// TIA Portal V17 export
// export: Created 2022-07-20T07:02:31.7533265Z, ExportSetting WithDefaults, DisplayName Totally Integrated Automation Portal, DisplayVersion V17, DisplayName TIA Portal Openness, DisplayVersion V17, DisplayName TIA Portal Version Control Interface, DisplayVersion V17, DisplayName SINAMICS Startdrive Advanced, DisplayVersion V17, DisplayName SINAMICS Startdrive G130, G150, S120, S150, SINAMICS MV, S210, DisplayVersion V17, DisplayName SINAMICS Startdrive G110M, G120, G120C, G120D, G120P, G115D, DisplayVersion V17, DisplayName STEP 7 Professional, DisplayVersion V17, DisplayName STEP 7 Safety, DisplayVersion V17, DisplayName WinCC Advanced, DisplayVersion V17
FUNCTION_BLOCK "FB11005_SheetEdgeDetection"   // FB11005, LAD
TITLE = Manage sheet edge detection
{ S7_Optimized_Access := 'TRUE' }
VERSION : 0.1
// stored: AutoNumber false, IsIECCheckEnabled false, IsRetainMemResEnabled false, MemoryReserve 100, SetENOAutomatically false, UDAEnableTagReadback false
   VAR_INPUT
      Enable { ExternalAccessible := 'False'; ExternalVisible := 'False'; ExternalWritable := 'False'} : Bool;
      Reset { ExternalAccessible := 'False'; ExternalVisible := 'False'; ExternalWritable := 'False'} : Bool;
      GapDrumSensor { ExternalAccessible := 'False'; ExternalVisible := 'False'; ExternalWritable := 'False'} : Real;
      GapBetweenSheet : Real;
   END_VAR
   VAR_OUTPUT
      Error { ExternalAccessible := 'False'; ExternalVisible := 'False'; ExternalWritable := 'False'} : Bool;
      ErrorSheetTooClose : Bool;
      WarningSheetTooClose : Bool;
      StartSheetPosition { ExternalAccessible := 'False'; ExternalVisible := 'False'; ExternalWritable := 'False'} : LReal;
      SheetDetected { ExternalAccessible := 'False'; ExternalVisible := 'False'; ExternalWritable := 'False'} : Bool;
      SheetGap : LReal;
      SensorActivated : Bool;
   END_VAR
   VAR_IN_OUT
      FilmDrumSensor : TO_MeasuringInput;
   END_VAR
   VAR
      R_TRIG_FilmDrumSensor { S7_SetPoint := 'True'} : R_TRIG;
      statFilmDrumPosition { S7_SetPoint := 'True'} : LReal;
      statFilmDrumPositionOld : LReal;
      statErrorMC : Bool;
      statJam : Bool;
      statOutfeedPosition : LReal;
      statStackerPosition : LReal;
      instMC_MEASURINGINPUT { S7_SetPoint := 'True'} : MC_MEASURINGINPUT;
   END_VAR
BEGIN

REGION Network 1 (SCL): Comments
   //==========================================================================================
   // SIEMENS SAS      RC-FR DI FA APC
   //------------------------------------------------------------------------------------------
   // Restrictions:    TIA V16 and more
   // Requirements:    S7-1500 + MGI library
   // Functionality:   This function block get position value of sheet edge 
   //------------------------------------------------------------------------------------------
   // Change log table:
   // Version      Date        Expert in charge    Changes applied
   // 01.00.01     09.06.2020  RTO                 First released version
   //==========================================================================================
END_REGION

REGION Network 2 (SCL): First Scan
   IF "FirstScan" THEN

       // Output
       #Error := FALSE;
       #SheetDetected := FALSE;
       #StartSheetPosition := 0.0;

       // Static
       #statFilmDrumPosition := 0.0;
       #statFilmDrumPositionOld := 0.0;
       #statErrorMC := FALSE;
       #statJam := FALSE;
       #statOutfeedPosition := 0.0;
       #statStackerPosition := 0.0;

   END_IF;
END_REGION

REGION Network 3 (SCL): Edge Signal Management
   REGION EDGE SIGNALS
       #R_TRIG_FilmDrumSensor(CLK := #FilmDrumSensor.InputState);
   END_REGION
END_REGION

REGION Network 4: Manage sensor acquisition
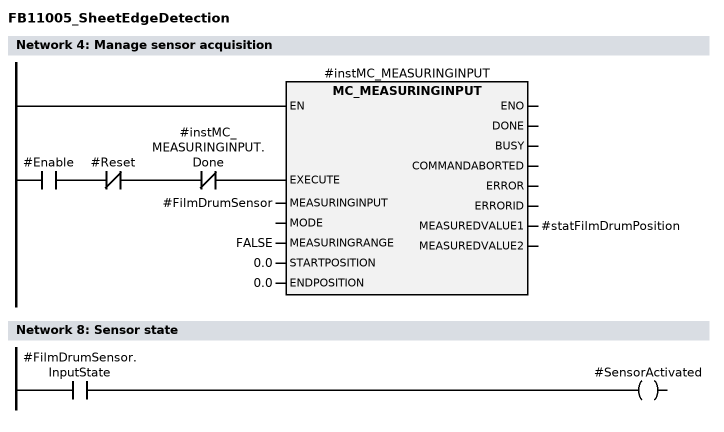
   RUNG wire#powerrail
      #instMC_MEASURINGINPUT.MC_MEASURINGINPUT(Execute := wire#w1, MeasuringInput := #FilmDrumSensor, Mode :=, MeasuringRange := FALSE, StartPosition := 0.0, EndPosition := 0.0, Done =>, Busy =>, CommandAborted =>, Error =>, ErrorId =>, MeasuredValue1 => #statFilmDrumPosition, MeasuredValue2 =>)
   END_RUNG
   RUNG wire#powerrail
      Contact( #Enable )
      I_Contact( #Reset )
      I_Contact( #instMC_MEASURINGINPUT.Done )
   END_RUNG wire#w1
   // the same network as SCL:
   #instMC_MEASURINGINPUT(Execute := #Enable AND NOT #Reset AND NOT #instMC_MEASURINGINPUT.Done,   // MC_MEASURINGINPUT
                          MeasuringInput := #FilmDrumSensor,
                          MeasuringRange := FALSE,
                          StartPosition := 0.0,
                          EndPosition := 0.0,
                          MeasuredValue1 => #statFilmDrumPosition);
END_REGION

REGION Network 5 (SCL): Manage sheet detection and position of synchronism
   IF #instMC_MEASURINGINPUT.Done THEN
       #SheetDetected := TRUE;
       #StartSheetPosition := #statFilmDrumPosition + #GapDrumSensor;
       #SheetGap := ABS(#statFilmDrumPosition - #statFilmDrumPositionOld);
       #statFilmDrumPositionOld := #statFilmDrumPosition;
   END_IF;

   IF #instMC_MEASURINGINPUT.Busy THEN
       #SheetDetected := FALSE;
   END_IF;

   IF #Reset THEN
       #SheetDetected := FALSE;
       #StartSheetPosition := 0.0;
   END_IF;
END_REGION

REGION Network 6 (SCL): Manage error
   IF #statErrorMC THEN
       #Error := TRUE;
   ELSIF #Reset THEN
       #Error := FALSE;
   END_IF;
END_REGION

REGION Network 7 (SCL): Manage measuring sheet gap and error too close

   IF #SheetGap > 0 THEN
       #ErrorSheetTooClose := #SheetGap < #GapBetweenSheet;
       #WarningSheetTooClose := #SheetGap < #GapBetweenSheet * 1.1;
   ELSE
       #ErrorSheetTooClose := FALSE;
       #WarningSheetTooClose := FALSE;
   END_IF;
END_REGION

REGION Network 8: Sensor state
   RUNG wire#powerrail
      Contact( #FilmDrumSensor.InputState )
      Coil( #SensorActivated )
   END_RUNG
   // the same network as SCL:
   #SensorActivated := #FilmDrumSensor.InputState;
END_REGION
END_FUNCTION_BLOCK
